FUNCTION_BLOCK CU050RecoverTask EXTENDS CUBaseRecover IMPLEMENTS ICUTask
VAR

END_VAR

Run();

(*~
	<docu>
		<summary>
			Main method of the sequener. Custom code needs to be placed here. The sequencer is executed by call of **Instance.Run()** method.
			This method is abstract, and it must be overridden in derived block.
		</summary>
	</docu>
~*)
METHOD PROTECTED Main : BOOL
(*

	RECOVER PROCESS 
	Following steps provide recover action for this controlled unit.
	Add components add write customized sequence according to your need.
*)

		
//
IF (Step(100, TRUE, '<#WAITING FOR START#>')) THEN
    //-------------------------------------    

    StepCompleteWhen(TRUE);
    //-------------------------------------
END_IF

//HERE  YOU CAN WRITE  WHAT IS NECESSARY 
//TO RECOVER AFTER INTERUPTED PROCESS.....

IF (Step(1000, TRUE, '<#RECOVER ANY COMPONENTS#>')) THEN
    //-------------------------------------    

    StepCompleteWhen(CurrentStep.Duration >= T#3000MS);
    //-------------------------------------
END_IF

IF (Step(30000, TRUE, 'RECOVER DONE')) THEN
    //-------------------------------------
		
        this^._done:=true;
		THIS^.Task.DoneWhen(TRUE);
		
   
    //-------------------------------------	
END_IF
END_METHOD

METHOD PUBLIC OnStart
SUPER^.OnStart();
Station.SuspendTask.Restore();
END_METHOD

PROPERTY Station : REFERENCE TO CU050
GET
VAR
    _station : POINTER TO CU050;
END_VAR
IF __QUERYPOINTER(Parent, _station) THEN // Check if _Parent is Station001
    Station REF= _station^;              // If the check is successful dereference a pointer. simlar to THIS^ or SUPER^
END_IF
END_GET
END_PROPERTY

END_FUNCTION_BLOCK

(* stored: Version 1.1.0.1
   POU CU050RecoverTask: Id {167883c5-19fc-4238-a4c6-db0af58e5eb1}, SpecialFunc None
   Method Main: Id {90d36f76-389d-4783-9499-5c8cab5881f9}
   Method OnStart: Id {a686f1d7-ba6d-4e4b-9de6-0ac9db7e1f93}
   Property Station: Id {a2ccd689-5dca-4fb9-8802-116e3438a474}
   Get Get: Id {808e1538-39da-43df-8cbc-792939f51b5f} *)
